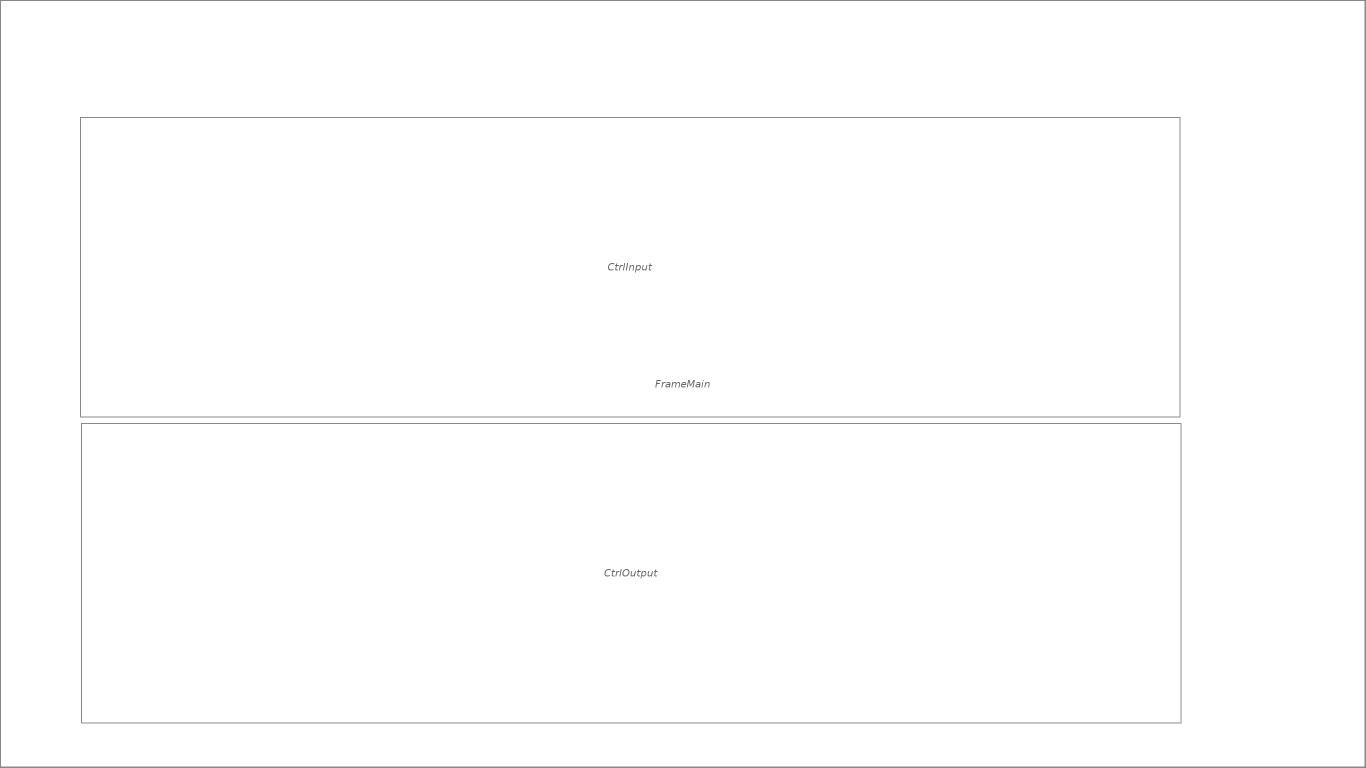
VISUALIZATION PageMonitor  // 1366x768
    Frame (0,0 1366x768)
        shows FrameMain()
    Frame (80,117 1100x300)
        shows CtrlInput(In := ADR(GVL_IO.I_Temp), SizeIn := Sizeof(GVL_IO.I_Temp), Enable := false, Ton := ADR(GVL_Data.stRecipe.arrInputTon), In_S := ADR(GVL.stShield_I))
    Frame (81,423 1100x300)
        shows CtrlOutput(In := ADR(GVL_IO.Q_Temp), SizeIn := sizeof(GVL_IO.Q_Temp), Enable := G_stSystem.stMode.bSetting, Ton := ADR(GVL_Data.stRecipe.arrOutputTon), In_S := ADR(GVL.stShield_Q))
END_VISUALIZATION

(* stored: Version 1.1.0.1, ProductVersion 3.1.4024.3
   Visu PageMonitor: Id {31385dff-1534-4d45-a4f9-d4fc843bcf47} *)
